INTERFACE I_StringBuilder

METHOD M_Append : I_StringBuilder
VAR_INPUT
	Value	: STRING(255);
END_VAR
END_METHOD

METHOD PUBLIC M_AppendBOOL  : I_StringBuilder
VAR_INPUT
	Value:			BOOL;
END_VAR
END_METHOD

METHOD PUBLIC M_AppendINT : I_StringBuilder
VAR_INPUT
	Value	: LINT;
END_VAR
END_METHOD

METHOD PUBLIC M_AppendREAL : I_StringBuilder
VAR_INPUT
	Value:		LREAL;
	nDecimals:	SINT;
END_VAR
END_METHOD

METHOD M_CopyTo : BOOL
VAR_INPUT
	Value:			ANY_STRING;
END_VAR
END_METHOD

METHOD M_Reset : I_StringBuilder
END_METHOD

METHOD PUBLIC M_ToString : String(255)
VAR_INPUT
END_VAR
END_METHOD

PROPERTY PUBLIC P_Length : Udint
GET
END_GET
END_PROPERTY

END_INTERFACE

(* stored: Version 1.1.0.1
   Itf I_StringBuilder: Id {df3d4a37-6b19-0224-3a23-50c560e48de6}
   Method M_Append: Id {ba3dc35a-00e3-0c07-0dfd-8c13ef431e5e}
   Method M_AppendBOOL: Id {7603f41d-77e0-0877-3137-edeb0957466d}
   Method M_AppendINT: Id {14f51f13-e329-0cde-0c9e-a7dc465a3499}
   Method M_AppendREAL: Id {f057156e-5dae-0fd8-10fe-cc573cd3ed43}
   Method M_CopyTo: Id {940c2d63-a99a-009b-232c-ea17ccc23948}
   Method M_Reset: Id {c51c1de9-e242-0e2e-15b4-007d70478885}
   Method M_ToString: Id {3d41c117-e4c2-0981-0e95-35260077a987}
   Property P_Length: Id {917505ca-54ce-03d7-1d45-2467135a7e41}
   Get Get: Id {9df562a0-8d74-0cfe-38db-8a1fcfe61f0c} *)
